{attribute 'qualified_only'}
VAR_GLOBAL
	



END_VAR

(* stored: Version 1.1.0.1, ProductVersion 3.1.4024.11
   GVL GVL: Id {cef261ee-0722-40ae-9d45-951d9804b073} *)
